Universal Robots URScript: SUB_141.script

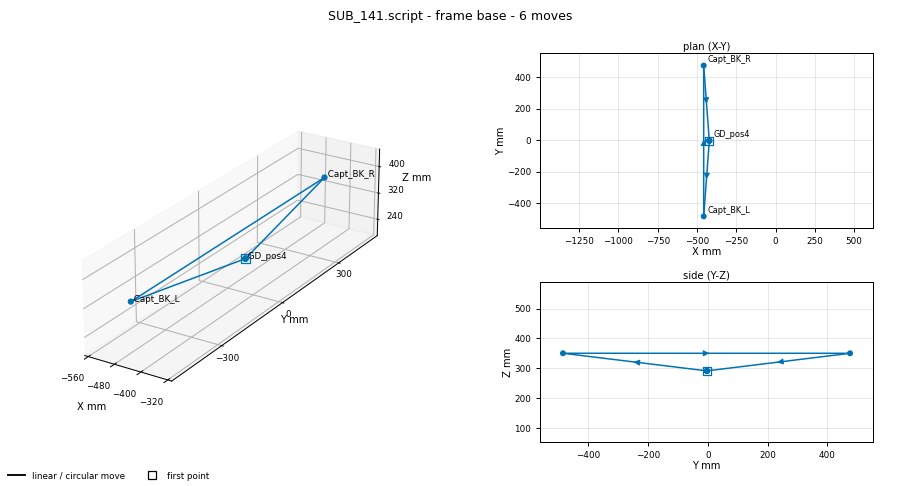
[picture p0: tool path of SUB_141.script in frame base, 6 of 6 moves have a stored position in this frame; points joined in program order, loops and branches not executed]
def SUB_141():
  global _hidden_verificationVariable=0
  set_tool_communication(False, 115200, 0, 1, 1.5, 3.5)
  set_tool_output_mode(0)
  set_tool_digital_output_mode(0, 1)
  set_tool_digital_output_mode(1, 1)
  set_tool_voltage(0)
  set_standard_analog_input_domain(0, 1)
  set_standard_analog_input_domain(1, 1)
  set_tool_analog_input_domain(0, 1)
  set_tool_analog_input_domain(1, 1)
  set_analog_outputdomain(0, 0)
  set_analog_outputdomain(1, 0)
  set_input_actions_to_default()
  set_runstate_gp_boolean_output_to_value(0, 3)
  set_target_payload(0.100000, [0.135000, 0.000000, 0.225000], [10.000000, 10.000000, 10.000000, 0.000000, 0.000000, 0.000000])
  set_safety_mode_transition_hardness(1)
  set_tcp(p[0.0,0.06,0.45,0.0,0.0,0.0])
  set_gravity([0.0, 0.0, 9.82])
  global isReCapt=False
  global Bucket_Z=[0, 0.7]
  global DistPillar=0
  global CandCnt=0
  global lr=1
  global ReCaptZ=0.05
  global forceval=p[0, 0, 0, 0, 0, 0]
  global CaptDepth=[0, 0, 0]
  global port=3000
  global isOnlyF=True
  global retX2=p[10000, 0, 0, 0, 0, 0]
  global socket_timeout=120
  global isSkipP=False
  global curpos=p[0, 0, 0, 0, 0, 0]
  global host="192.168.1.2"
  global is_popup=False
  global CaptZOffset=0
  global isGoHome=True
  global i_pos2=p[0.71903, -0.14046, 0.13075, 1.99335, -2.11497, -0.36069]
  global i_pos1=p[0.71664, -0.14067, 0.1303, 1.9903, -2.11284, -0.36439]
  global pBucket=[p[10000, 0, 0, 0, 0, 0], p[10000, 0, 0, 0, 0, 0], p[0, 0, 0, 0, 0, 0]]
  global CaptStepZ=0.08
  global CaptIndex=[0, 0, 0]
  global CaptStepX=0.432
  global pBucketM=p[-0.80141, -0.42542, 0.2879, 0, 0, 1.55713]
  global socket_name="vt"
  global rovi_err=0
  global SubPrgResult=100
  global CurrPos=p[0.00284, -0.38817, 0.46932, 0.06387, -3.14074, 0.00007]
  global CurrPos_p=p[0.00031, -0.32825, 0.01932, 0.06387, -3.14074, 0.00007]
  global ForceStartZ=0.4352
  global CutOffZ=0.08
  global HomeDistTh=0.05
  global RBDistTh=0.05
  global RBRadiusTh=0.3
  global RBXTh=[-0.5, 0.5]
  global RBYTh=[-0.8, 1]
  global RBZTh=[-0.1, 0.1]
  global Sub3100_ZMax=0.74
  global ForceStartX=-0.98868
  global Sub3100_aRot=0.2
  global Sub3100_d=0.3
  global Sub3100_Option=2
  global Sub3100_a=0.2
  global Sub3100_XdV=0.1
  global Sub3100_XdRot=8
  global ZoneDistTh=0.05
  global ZoneRadiusTh=0.3
  global ZoneXTh=[-0.5, 0.5]
  global ZoneYTh=[-0.8, 1]
  global ZoneZTh=[-0.1, 0.1]
  global BucketWidth=0.95
  global ZoneBucketGap=0.1
  global ZoneHomeX=[-0.2, 0.2]
  global UnloadZ=0.05
  global CaptPos=p[0.4274, -0.37367, 0.0721, 3.13247, 0.05506, 0.01735]
  global BucketUpperPos=p[0.4274, -0.37367, 0.0721, 3.13247, 0.05506, 0.01735]
  global Sub3100_GPII18=2
  global Bucket=p[0.32604,0.49174,0.0,-1.882900624652718E-5,2.8304179127934987E-5,-1.593185305749222]
  global BucketM=p[0.32604,0.49174,0.0,2.2353980716304163E-16,-3.5868426080024975E-16,-1.5931853071795856]
  global CaptPoint_C=p[-0.4219337985373468,-0.003168602281063755,0.36,-2.1962364319979395,-2.2439316084554193,-0.02184884826814999]
  global CaptPoint_C2=p[0.32796661698047924,-0.010768520544682924,0.01931625281283378,2.2288103429550152,-2.213636886217198,8.598462540813273E-5]
  global CaptPoint_L1=p[-0.42193494849366175,-0.2,0.36,-2.1962086037526616,-2.243896582262281,-0.02199725151102503]
  global CaptPoint_L2=p[0.327894307417917,-0.010799940826224014,0.01928712668893995,2.087717047309385,-2.0736781215133306,0.27365839887453103]
  global CaptPoint_R1=p[-0.4219551896101372,0.3,0.36,-2.1960823751566156,-2.243954123514977,-0.021863042557794844]
  global CaptPoint_R2=p[0.327926308680866,-0.010795166414457658,0.019300245403843563,-2.1186306375223185,2.1040550557443427,0.22023197678473694]
  global Capt_1BK_L=p[-0.4574214308482636,-0.48457071473611046,0.3504487959434708,-2.1962343446504526,-2.243967222238911,-0.021809195357489434]
  global Capt_1BK_R=p[-0.4574597285646511,0.4755214243904677,0.35039311859649847,-2.196330286580149,-2.2438949166739053,-0.021738621025254933]
  global Capt_1BK_pos1=p[-0.4218793038724447,-0.003154429464978058,0.2915499891144615,-2.1963422029204875,-2.2438663520270015,-0.02197160668673838]
  global Capt_1BK_pos2=p[-0.42187829024618434,-0.0031710253373066375,0.29156503858953065,-2.196324918349679,-2.2439040699490773,-0.021928444416953782]
  global Capt_2BK_L=p[0.42186661528427194,0.4254738068040517,0.35042275762909847,2.239156309475874,-2.1837044610999294,0.002643817066643282]
  global Capt_2BK_R=p[0.4218208572756906,-0.5427676723257963,0.350372239919558,2.2392697861179327,-2.183553596194912,0.002410470905346486]
  global Capt_2BK_pos1=p[0.42193501458435656,0.004742683868356356,0.35045865974037793,2.2391012408536453,-2.1839704655717003,0.002677867056024068]
  global Capt_2BK_pos2=p[0.421903984494575,0.004707988774967922,0.35045218900915065,2.239114367170047,-2.183895515396197,0.002684056681074047]
  global Capt_GD_M=p[-0.004053197679954899,-0.25261725691632436,-0.01970497430780127,0.0332779454553888,-3.140179196376707,-0.0034093680964018282]
  global HomePointL=p[-0.36789,-0.5117344641471838,0.78,-0.6278857271586024,3.0680899128661667,-8.649957362498864E-4]
  global PickPos=p[0.10830682331105715,-1.3709505888096256,-0.18404188875951455,-0.00622194000158997,2.880236948927292,-0.00383636509397631]
  global Solve=p[-0.00368,-0.0021000000000000003,0.25739999999999996,0.0,0.0,0.0]
  global TEST=p[0.1,0.0,0.2,0.0,0.0,0.0]
  global UF=p[0.0,0.0,0.0,0.0,0.0,0.0]
  global g1CV_1_M=p[0.29093319989156785,-0.9405344885124904,-0.08686754932079166,1.9884186265311852,2.2323374792844253,0.1524643645929425]
  global g1CV_posL1=p[0.05028133628211688,-0.4526481033729615,0.1221845548632916,-2.213335080948508,-2.1937561336067057,-0.3280056759040735]
  global g1CV_posR1=p[0.03743870476062511,-0.53119407812668,0.11301901343688614,2.073418671558482,2.153257467049566,0.11656306439039889]
  global g1GD_pos1=p[0.06841781024889843,-0.5456037307108855,0.367146167315866,2.4108578981103275,1.7957834606331096,0.12544942012730473]
  global g1GD_pos2=p[-0.38705506163240566,-0.3905161646272917,0.3670805000411974,2.9334800678601534,0.5562338866571123,0.025147235284150155]
  global g1GD_pos3=p[-0.614523200343285,-0.009392732880809615,0.3783325239377683,2.0687271625579515,2.17319336139756,0.21682066343437634]
  global g1GD_pos4=p[-0.4351564513137486,0.028155221259926276,0.13086718327275837,2.2072871432536783,2.2307343865376095,-0.0018307218179379997]
  global g1GD_pos5=p[-0.8151645021025727,-0.01706756320728201,0.08179601375099321,2.212895896456039,2.218350348620789,0.019350113017735118]
  global g1GD_posL1=p[-0.08276848269606216,-0.3996147100031649,0.1488453551331823,2.286527078917204,1.8420745504477611,0.33698451773695576]
  global g1GD_posL2=p[-0.3253977027403738,-0.3024804624281039,0.16332814085945146,2.72312820760317,0.9631021078169197,0.32447452035226126]
  global g1GD_posL3=p[-0.6791033397183219,0.06787475590683856,0.16337212788108813,2.1383125299263996,2.086116032377724,0.4536080263755059]
  global g1GD_posR1=p[-0.09893370538053747,-0.4999608954567234,0.14329885217724153,2.43311852414254,1.4238397520832589,0.08559216753941556]
  global g1GD_posR2=p[-0.3729565201882258,-0.3752983669473301,0.143299052800563,2.6951655216297596,0.8130506811102118,-0.02387549506099888]
  global g1GD_posR3=p[-0.7385929502572233,-0.029472684480355026,0.1499650660949685,2.0484522752014467,1.9493695704119496,0.18368227556562683]
  global g2CV_1_M=p[0.2880593256931911,-0.933809998732841,-0.08698643380656113,2.0727630257838867,2.230596497566155,0.15036691287620893]
  global g2CV_posL1=p[0.3409386496330911,-0.4656338066361442,0.1250074988128972,2.209372209162659,2.1945371304665926,0.3160714960040194]
  global g2CV_posR1=p[0.3400736278759575,-0.531334269888987,0.1183415684753657,2.07314649492589,2.1532617466521136,0.11638666128062146]
  global g2GD_pos1=p[0.3390086633742754,-0.5203839341398588,0.22258,2.022696172282159,2.259224887850344,0.09811005079237367]
  global g2GD_pos2=p[0.4140891885236144,0.14850105084950693,0.1582916370575993,-0.10302503203970696,3.1008909166713883,0.18748967846962497]
  global g2GD_pos3=p[0.32377086541216454,-0.01023215987367155,0.15821240334102793,2.279746475463588,-2.06129961332614,-0.16578334012307952]
  global g2GD_pos4=p[0.7398823109797592,-0.026643494293930835,0.22255839224074236,2.162283599874437,-2.168919538925757,-0.13861635932587069]
  global g2GD_pos5=p[0.22271243238356278,-0.026679271241024524,0.22257782526136982,1.3056143664331146,-2.8077458860488136,-0.17177240522535248]
  global gCV_11_M=p[0.3028468774759881,-0.9375366886748661,-0.09782511939875749,1.9971971468330036,2.0934336167121885,0.3604928446251781]
  global gCV_12_M=p[0.34776610649632045,-0.9364202289953052,-0.09784932758070936,1.9972781240484352,2.0934384510830295,0.3604701319279358]
  global gCV_13_M=p[0.43083047728791135,-0.9363258116427577,0.028711300566433673,1.9972504931093251,2.0935710325846095,0.3605630596092243]
  global gCV_14=p[0.35645641620611146,-0.8914305774826713,-0.17737239800677018,2.1506886654737776,2.1461343800624295,0.40986447399780934]
  global gCV_15=p[0.4370373250739419,-0.891408661166693,-0.1773997714481486,2.1507483614991094,2.1461657601704176,0.40983132876462236]
  global gCV_16=p[0.4597123429384979,-0.8913837618729653,-0.03599504377258328,2.1506156333226136,2.1462305295546718,0.4099109158136618]
  global gCV_17=p[0.037528034463104695,-0.6904892259828748,-0.12243237639232962,-0.12012393052395552,2.832430475095037,0.48967048060305135]
  global gCV_18=p[0.03600103065313248,-0.6368623043127666,-0.12241687036449483,-0.12010351348807546,2.832474314609516,0.48970816626953567]
  global gCV_2_M=p[0.2909259851094176,-0.9405632657218349,0.07217586581493451,1.9883998690824036,2.232303337331875,0.15240099649164607]
  global gCV_3_M=p[0.29099390607376485,-0.6570558385379063,0.0722153583041818,1.9884242634571576,2.2321538498123994,0.15249643504377583]
  global gCV_5=p[0.045776199142861046,-0.9791473230816141,0.8415069045351792,2.0229894037377316,2.080009888728606,0.35618099403901887]
  global gCV_pos5=p[0.3400172856834047,-0.9722754606605235,-0.18287928563575456,2.073394561413637,2.1531827558666565,0.11639000988241816]
  global gGD_100_1LM=p[0.04146780808756359,-0.6870904124925177,-0.1232943093634104,-0.006305250057386166,-2.863965809273829,-0.5082528300185785]
  global gGD_1_LM=p[0.039828597127514714,-0.6781969854050135,-0.12198496009202514,-0.035987858392923795,2.830752931487768,0.5274559890082169]
  global gGD_1_M=p[0.04223412605599862,-0.6762907291217815,-0.12305211139062167,0.03206414188010415,3.0719576115730227,0.5678560916913992]
  global gGD_1_MM=p[0.03527332731929103,-0.7200324399236822,-0.12309145975746483,-0.05946537723025455,3.087281488106925,0.5412792107775745]
  global gGD_1_RM=p[0.044824714971060706,-0.6786804080355537,-0.12465669282958386,-0.09848782436012833,-2.854704518703978,-0.5230067998162747]
  global gGD_200_2LM=p[0.04175812558137225,-0.6358261219893102,-0.12285474020423298,-0.006257718193554584,-2.863964784148567,-0.5084621939645108]
  global gGD_2_LM=p[0.039831971231659546,-0.6353194260198303,-0.12200751601005971,-0.036099546068508924,2.830809185470081,0.52731796109078]
  global gGD_2_M=p[0.042191660627195246,-0.635754045905828,-0.12312962051191373,0.03192332016161312,3.0719623350853844,0.5679093611320986]
  global gGD_2_RM=p[0.044795235627329705,-0.6336331294114242,-0.12463856522096584,-0.09855677972998968,-2.8547026274584586,-0.522938600214494]
  global gGD_300_3LM=p[0.04182050265947469,-0.6066076810742604,-0.03602288107395374,-0.006290924000441408,-2.8640915241774816,-0.5083501301248439]
  global gGD_3_LM=p[0.039836850432748136,-0.5755330743649689,-0.010235964588677704,-0.03615378224605123,2.8308405562482424,0.5271952258447209]
  global gGD_3_M=p[0.04221104672013029,-0.5661292175118147,0.002580299638146877,0.03178620336833174,3.071951282137014,0.5679299882450841]
  global gGD_3_RM=p[0.04485568823805332,-0.5667893626574417,-0.012456252830579384,-0.09850858677456549,-2.854716139592613,-0.5230996025040573]
  global gGD_400_1RM=p[0.03765496539143813,-0.6905733748742057,-0.12240702670509729,-0.12009639012349203,2.8324503628258273,0.48945657912051843]
  global gGD_4_LM=p[-0.050697518013391604,-0.4788149830819543,0.04525080740157289,-0.14673385744666134,2.827848291285266,0.5267055795817903]
  global gGD_4_RM=p[0.10921584432919978,-0.48073334437858256,0.06990685637741062,0.016338390530391603,-2.862804566994448,-0.49861203356258266]
  global gGD_500_2RM=p[0.0364038044475721,-0.6361408639594927,-0.1228896102948493,-0.12001814478849077,2.8324363686538967,0.4895422385690364]
  global gGD_600_3RM=p[0.03597788557419286,-0.6039591135870097,-0.03251312847845622,-0.12016380804709932,2.832584395249392,0.4895204315491753]
  global gGD_M_20=p[0.03524102305764369,-0.704963855446233,-0.12310321086399345,-0.05961230604660993,3.0873078767639504,0.5414261100507907]
  global gGD_M_30=p[0.03527181411394771,-0.6949613298581867,-0.12309199448652725,-0.05962447301074729,3.087287038166274,0.5412100180254447]
  global gGD_M_40=p[0.035236425258241534,-0.6834410208824955,-0.12309554834290798,-0.05953064339288712,3.087315110349415,0.5412921265180426]
  global gHome_Position=p[3.053061697190075E-4,-0.3281132156787397,0.01930332806480972,0.0637196994340987,-3.140722020313799,-3.2847660283345163E-4]
  rtde_set_watchdog("speed_slider_mask", 10.0, "ignore")
  # begin: URCap Installation Node
  #   Source: Ethernet/IP I/O Monitor URCap, 1.0.0,
  #   Type: Ethernet/IP I/O Monitor
  conn = rpc_factory("xmlrpc", "http://127.0.0.1:" + to_str(61101) + "/RPC2")

  def show_monitor():
    return conn.eip_monitor.show()
  end
  # end: URCap Installation Node
  step_count_3bdac028_a61b_406d_9d29_047d8a4f5e6b = 0.0
  thread Step_Counter_Thread_e78790e0_9fd0_4dbc_bed3_2ed3a53882eb():
    while (True):
      step_count_3bdac028_a61b_406d_9d29_047d8a4f5e6b = step_count_3bdac028_a61b_406d_9d29_047d8a4f5e6b + 1.0
      sync()
    end
  end
  run Step_Counter_Thread_e78790e0_9fd0_4dbc_bed3_2ed3a53882eb()
  while (True):
    $ 2 "ロボットプログラム"
    $ 3 "INITIALIZE"
    $ 4 "荷重の設定: k10"
    set_target_payload(0.100000, [0.135000, 0.000000, 0.225000], [10.000000, 10.000000, 10.000000, 0.000000, 0.000000, 0.000000])
    $ 5 "設定"
    set_tcp(p[0.14,0.0,0.0,0.0,0.0,0.0])
    $ 6 "If文 (GPII_WorkPosNo≟1)"
    if ((read_input_integer_register(4) == 1)):
      $ 7 "GD_pos4:=Capt_2BK_pos1"
      global GD_pos4=Capt_2BK_pos1
      $ 8 "GD_pos5:=Capt_2BK_pos2"
      global GD_pos5=Capt_2BK_pos2
      $ 9 "Capt_BK_L:=Capt_2BK_L"
      global Capt_BK_L=Capt_2BK_L
      $ 10 "Capt_BK_R:=Capt_2BK_R"
      global Capt_BK_R=Capt_2BK_R
    else:
      $ 11 "ElseIf (GPII_WorkPosNo≟2)"
      if ((read_input_integer_register(4) == 2)):
        $ 12 "GD_pos4:=Capt_1BK_pos1"
        global GD_pos4=Capt_1BK_pos1
        $ 13 "GD_pos5:=Capt_1BK_pos2"
        global GD_pos5=Capt_1BK_pos2
        $ 14 "Capt_BK_L:=Capt_1BK_L"
        global Capt_BK_L=Capt_1BK_L
        $ 15 "Capt_BK_R:=Capt_1BK_R"
        global Capt_BK_R=Capt_1BK_R
      end
    end
    $ 16 "HOME"
    $ 17 "MoveJ"
    $ 19 "GD_pos4" "breakAfter"
    set_tcp(p[0.0,0.06,0.45,0.0,0.0,0.0])
    movej(GD_pos4, a=0.5235987755982988, v=1.2217304763960306)
    $ 20 "MoveL"
    $ 21 "GD_pos5" "breakAfter"
    movel(GD_pos5, a=0.07, v=0.2)
    $ 23 "ROVI_RECIPE"
    $ 24 "recipe_bucket:=GPII_BucketNo"
    global recipe_bucket=read_input_integer_register(3)
    $ 25 "If文 ( not ROVI_RECIPE(recipe_bucket))"
    if ((  not  ROVI_RECIPE(recipe_bucket))):
      $ 26 "SubPrgResult:=rovi_err"
      global SubPrgResult=rovi_err
      $ 27 "待機: 999999.0"
      sleep(999999.0)
    end
    $ 28 "ROVI_RESET"
    $ 29 "If文 ( not ROVI_RESET())"
    if ((  not  ROVI_RESET())):
      $ 30 "SubPrgResult:=rovi_err"
      global SubPrgResult=rovi_err
      $ 31 "待機: 999999.0"
      sleep(999999.0)
    end
    $ 32 "ROVI_CAPTURE_1"
    $ 33 "MoveL"
    $ 34 "Capt_BK_L" "breakAfter"
    set_tcp(p[0.0,0.06,0.45,0.0,0.0,0.0])
    movel(Capt_BK_L, a=0.07, v=0.2)
    $ 35 "待機: 2.0"
    sleep(2.0)
    $ 36 "If文 ( not ROVI_CAPTURE())"
    if ((  not  ROVI_CAPTURE())):
      $ 37 "SubPrgResult:=rovi_err"
      global SubPrgResult=rovi_err
      $ 38 "待機: 999999.0"
      sleep(999999.0)
    end
    $ 39 "ROVI_CAPTURE_2"
    $ 40 "MoveL"
    $ 41 "Capt_BK_R" "breakAfter"
    set_tcp(p[0.0,0.06,0.45,0.0,0.0,0.0])
    movel(Capt_BK_R, a=0.07, v=0.2)
    $ 42 "待機: 2.0"
    sleep(2.0)
    $ 43 "If文 ( not ROVI_CAPTURE())"
    if ((  not  ROVI_CAPTURE())):
      $ 44 "SubPrgResult:=rovi_err"
      global SubPrgResult=rovi_err
      $ 45 "待機: 999999.0"
      sleep(999999.0)
    end
    $ 46 "ROVI_SOLVE"
    $ 47 "retX2:=ROVI_SOLVE()"
    global retX2=ROVI_SOLVE()
    $ 48 "If文 (retX2[0]≟10000.)"
    if ((retX2[0] == 10000.)):
      $ 49 "SubPrgResult:=rovi_err"
      global SubPrgResult=rovi_err
      $ 50 "待機: 999999.0"
      sleep(999999.0)
    end
    $ 51 "HOME"
    $ 52 "MoveL"
    $ 53 "GD_pos5" "breakAfter"
    set_tcp(p[0.0,0.06,0.45,0.0,0.0,0.0])
    movel(GD_pos5, a=0.07, v=0.25)
    $ 54 "GD_pos4" "breakAfter"
    set_tcp(p[0.0,0.06,0.45,0.0,0.0,0.0])
    movel(GD_pos4, a=0.07, v=0.25)
  end
end
